PROGRAM P_4Packing
VAR
	nState: INT;
	
	//Timers
	fbTimerGrabX : TON;
	fbTimerGrabY : TON;
	fbTimerGrabZ : TON;
	fbTimerGrab : TON;
	fbTimerLift : TON;
	fbTimerDrop1 : TON;
	fbTimerDrop2 : TON;
	fbTimerMoving2 : TON;
	fbTimerMoving3 : TON;
	fbTimerMovingLoad : TON;
	fbTimerWaiting : TON;
	fbTimerEmitPal: TON;
	
	iCounterTrig: R_trig;
	
END_VAR
VAR CONSTANT
	//Here we define our constant where we want the different positon to be. This is instead of making steps you can call this fixed steps.
	Standby: 	INT:=00;
	GrabX:		INT:=10;
	GrabY:		INT:=11;
	GrabZ:		INT:=12;
	Grab:		INT:=13;
	Lift:		INT:=15;
	Drop1:		INT:=20;
	Drop2:		INT:=21;
	Moving1    : INT := 30;
	Moving2    : INT := 31;
	Moving3    : INT := 32;
	MovingStop : INT := 22;
	AtLoad:		INT:=35;	
	Waiting    : INT := 40;
	Stopping   : INT := 50;
	Resetting  : INT := 60;
	Estop      : INT := 99;
		
END_VAR

// This is our fourth program is where we count the anount of boxes that have been put together  and the second xyz arm will pick up the box 
// and place it on the pallet.

iCounterTrig(CLK:=FIO.bPP_PosRais_Base);  //define a trigger so we can use it to count the amount of boxes that have been put together.  

IF iCounterTrig.Q THEN                    //box counter
	FIO.iEbCounter:=FIO.iEbCounter+1;
END_IF


 
CASE nState OF
	
	Standby:      //the sensor is true when there are a box and a palled will emit 
		IF  FIO.bOutPaSens=TRUE THEN
			FIO.bScEmitPallet:=TRUE;	
			nState:=GrabX;		
		END_IF	
				

	GrabX:		//we move the XYZ arm in the X position 
		IF FIO.bOutPaSens=TRUE THEN    
			FIO.rOutPaMoveX:=4.5;
			fbTimerGrabX(IN:=TRUE,PT:=T#1S);	
			IF fbTimerGrabX.Q THEN
				fbTimerGrabX(IN:=FALSE); 
				nState:=GrabY;
			END_IF	
		END_IF

	GrabY:	//we move the XYZ arm in the Y position 
		IF FIO.rOutPaMoveX=4.5 THEN 
			FIO.rOutPaMoveY:=9.5;
			fbTimerGrabY(IN:=TRUE,PT:=T#1S);	
			IF fbTimerGrabY.Q THEN
				fbTimerGrabY(IN:=FALSE); 
				nState:=GrabZ;
			END_IF	
		END_IF
	
	GrabZ:  //we move the XYZ arm in the Z position 
		IF FIO.rOutPaMoveY=9.5 THEN 
			FIO.rOutPaMoveZ:=8.5;
			FIO.bOutPaToolRot:=TRUE;
			fbTimerGrabZ(IN:=TRUE,PT:=T#2S);	
			IF fbTimerGrabZ.Q THEN
				fbTimerGrabZ(IN:=FALSE); 
				nState:=Grab;
			END_IF				
		END_IF
	
	Grab:   //we here we turn the grab on so it can pick up a box
		IF FIO.bOutPaBoxDetected=TRUE THEN
			FIO.bOutPaGrab:=TRUE;
			fbTimerGrab(IN:=TRUE,PT:=T#1S);
			 IF fbTimerGrab.Q THEN
				fbTimerGrab(IN:=FALSE);
				nState:=Lift; 
		 	END_IF
		END_IF	
		
	Lift:    //here we lift the box
		IF FIO.bOutPaGrab=TRUE THEN
			FIO.rOutPaMoveZ:=0;
			fbTimerLift(IN:=TRUE,PT:=T#1S);
			 IF fbTimerLift.Q THEN
				fbTimerLift(IN:=FALSE);
				nState:=Drop1;
		 	END_IF					
		END_IF	

	Drop1:  // here move in Y axes so it is almost in the middle of the pallet
		IF FIO.rOutPaMoveZ=0 THEN
			FIO.rOutPaMoveY:=1.5;
			fbTimerDrop1(IN:=TRUE,PT:=T#1S);
			 IF fbTimerDrop1.Q THEN
				fbTimerDrop1(IN:=FALSE);
				nState:=Drop2;
		 	END_IF
		END_IF	
		
	Drop2:  //here we move the arm in Z position where we lower the har closer to the pallet and then we drop the box
		IF FIO.bOutPaGrab=TRUE THEN
			FIO.rOutPaMoveZ:=10;
			fbTimerDrop2(IN:=TRUE,PT:=T#1S);
			 IF fbTimerDrop2.Q THEN
				fbTimerDrop2(IN:=FALSE);
				FIO.bOutPaGrab:=FALSE;
				nState:=Waiting;;
		 	END_IF	
		END_IF


		
//----------------------------------------------------------------------------//

	Waiting:
			nState:=Standby;
		
			
		
//----------------------------------------------------------------------------//


	ELSE
		nState:=9999;	
END_CASE

END_PROGRAM

(* stored: Version 1.1.0.1, ProductVersion 3.1.4024.3
   POU P_4Packing: Id {44301db5-00b1-4ee0-9258-716fda2a1772}, SpecialFunc None *)
